# EPICS autosave request: softGlueApp/Db/UpDnCntr_settings.req
$(P)$(H)UpDnCntr-$(N)_CLOCK_Signal
$(P)$(H)UpDnCntr-$(N)_UPDOWN_Signal
$(P)$(H)UpDnCntr-$(N)_ENABLE_Signal
$(P)$(H)UpDnCntr-$(N)_CLEAR_Signal
$(P)$(H)UpDnCntr-$(N)_LOAD_Signal
$(P)$(H)UpDnCntr-$(N)_OUT_Signal
$(P)$(H)UpDnCntr-$(N)_PRESET
